// TIA Portal V19 export
DATA_BLOCK "MFG TRANSFER CYCLE DB"   // DB74
{ S7_Optimized_Access := 'TRUE' }
// stored: MemoryReserve 100
   VAR RETAIN
      TRANSFER : Struct
         "TRANSFER START" : Bool;
         "TRANSFER STOP" : Bool;
         "TRANSFER OVER" : Bool;
         "TRANSFER BUFF" : Struct
            "MFG TO STORAGE-1 WITH INLINE HOMO" : Int;
            "MFG TO STORAGE-1 WITH INLINE FILTER PRES" : Int;
            "MFG TO STORAGE-2 WITH INLINE HOMO" : Int;
            "MFG TO STORAGE-2 WITH INLINE FILTER PRES" : Int;
            "MFG TO STORAGE-3 WITH INLINE HOMO" : Int;
            "MFG TO STORAGE-3 WITH INLINE FILTER PRES" : Int;
         END_STRUCT;
         SELECT : Struct
            "MFG TO STORAGE-1 WITH INLINE HOMO" : Bool;
            "MFG TO STORAGE-1 WITH INLINE FILTER PRES" : Bool;
            "MFG TO STORAGE-2 WITH INLINE HOMO" : Bool;
            "MFG TO STORAGE-2 WITH INLINE FILTER PRES" : Bool;
            "MFG TO STORAGE-3 WITH INLINE HOMO" : Bool;
            "MFG TO STORAGE-3 WITH INLINE FILTER PRES" : Bool;
            "SELECT BUFF" : Int;
         END_STRUCT;
      END_STRUCT;
      "SET PARAMETER" : Struct
         "MFG TO STORAGE-1 WITH INLINE HOMO" : Real;
         "MFG TO STORAGE-1 WITH INLINE FILTER PRES" : Real;
         "MFG TO STORAGE-2 WITH INLINE HOMO" : Real;
         "MFG TO STORAGE-2 WITH INLINE FILTER PRES" : Real;
         "MFG TO STORAGE-3 WITH INLINE HOMO" : Real;
         "MFG TO STORAGE-3 WITH INLINE FILTER PRES" : Real;
         "SET TIME" : Struct
            "MFG TO STORAGE-1 WITH INLINE HOMO" : Int;
            "MFG TO STORAGE-1 WITH INLINE FILTER PRES" : Int;
            "MFG TO STORAGE-2 WITH INLINE HOMO" : Int;
            "MFG TO STORAGE-2 WITH INLINE FILTER PRES" : Int;
            "MFG TO STORAGE-3 WITH INLINE HOMO" : Int;
            "MFG TO STORAGE-3 WITH INLINE FILTER PRES" : Int;
         END_STRUCT;
         RPM : Struct
            "MFG TO STORAGE-1 WITH INLINE HOMO" : Real;
            "MFG TO STORAGE-1 WITH INLINE FILTER PRES" : Real;
            "MFG TO STORAGE-2 WITH INLINE HOMO" : Real;
            "MFG TO STORAGE-2 WITH INLINE FILTER PRES" : Real;
            "MFG TO STORAGE-3 WITH INLINE HOMO" : Real;
            "MFG TO STORAGE-3 WITH INLINE FILTER PRES" : Real;
         END_STRUCT;
      END_STRUCT;
      "PV PARAMETER" : Struct
         "MFG TO STORAGE-1 WITH INLINE HOMO" : Real;
         "MFG TO STORAGE-1 WITH INLINE FILTER PRES" : Real;
         "MFG TO STORAGE-2 WITH INLINE HOMO" : Real;
         "MFG TO STORAGE-2 WITH INLINE FILTER PRES" : Real;
         "MFG TO STORAGE-3 WITH INLINE HOMO" : Real;
         "MFG TO STORAGE-3 WITH INLINE FILTER PRES" : Real;
         "PV TIME" : Struct
            "MFG TO STORAGE-1 WITH INLINE HOMO" : Int;
            "MFG TO STORAGE-1 WITH INLINE FILTER PRES" : Int;
            "MFG TO STORAGE-2 WITH INLINE HOMO" : Int;
            "MFG TO STORAGE-2 WITH INLINE FILTER PRES" : Int;
            "MFG TO STORAGE-3 WITH INLINE HOMO" : Int;
            "MFG TO STORAGE-3 WITH INLINE FILTER PRES" : Int;
         END_STRUCT;
      END_STRUCT;
   END_VAR
BEGIN
END_DATA_BLOCK
